{attribute addProperty BoxType "EL3041-0000-0017"}
{attribute addProperty Id "AI_StandardAT %I*AI_Standard_B51B79FC8110.1250WcStateAT %I*WcState_F855686C1620InfoDataAT %I*InfoData_BC63D37F80100"}
{attribute addProperty CRC "368140935"}
{attribute addProperty SizeInBites "177"}
{attribute addProperty SizeInBytes "22.125"}
TYPE EL3041_4607B8C0 :
STRUCT
	{attribute addProperty Name "AI_Standard"}
	AI_Standard : AI_Standard_B51B79FC;
	{attribute addProperty Name "WcState"}
	WcState : WcState_F855686C;
	{attribute addProperty Name "InfoData"}
	InfoData : InfoData_BC63D37F;
END_STRUCT
END_TYPE

(* stored: Version 1.2.0.0, ProductVersion 3.1.4024.9
   DUT EL3041_4607B8C0: Id {7d7c531c-1233-42e4-bbd2-4f26b2feaae2} *)
